// TIA Portal V20 export
TYPE "HMI_MotSpdL"
   STRUCT
      Spd1Man : Bool := FALSE;   // 1=Start: Speed1 Command in Manual Mode
      Spd2Man : Bool := FALSE;   // 1=Start: Speed2 Command in Manual Mode
      StopMan : Bool := FALSE;   // 1=Stop: Stop Command in Manual Mode
      AutModOp : Bool := FALSE;   // 1=Auto Mode: Auto Mode by Operator
      ManModOp : Bool := TRUE;   // 1=Manual Mode: Manual Mode by Operator
      LocalLi : Bool;   // 1=Local Mode: Local Operation by Field Signal
      LocalOp : Bool := FALSE;   // 1=Local Mode: Local Operation by Operator
      OosOp : Bool := FALSE;   // 1=Oos Mode: Oos Mode by Operator
      Spd1Local : Bool;   // 1=Start Local: Field Speed1 Start Signal
      Spd2Local : Bool;   // 1=Start Local: Field Speed2 Start Signal
      StopLocal : Bool;   // 1=Stop Local: Field Stop Signal
      Monitor : Bool := TRUE;   // 1=Monitor ON, 0=Monitor OFF: Feedback Monitor
      MonTiStatic : Real := 3.0;   // Monitoring Time of Feedback [s]
      MonTiDynamic : Real := 3.0;   // Monitoring Time of Feedback on starting or on change in control output [s]
      MonTiDyStop : Real := 3.0;   // Monitoring Time of Feedback on stopping in control output [s]
      RapidStp : Bool := FALSE;   // 1 = Motor Rapid Stop command
      RstOp : Bool := FALSE;   // Operator Reset Signal
      Permit_ST : Byte := BYTE#16#FF;   // Permit Signal Status
      PermSp2 : Bool := true;   // 1= Activation Speed2 is allowed, 0= Not allowed
      PermSp2_ST : Byte := BYTE#16#FF;   // PermSp2 Signal Status
      Intlock_ST : Byte := BYTE#16#FF;   // Interlock Signal Status
      IntlSp2 : Bool := true;   // 0= Intlock Speed2 is active, 1= Not active
      IntlSp2_ST : Byte := BYTE#16#FF;   // IntlSp2 Signal Status
      Protect_ST : Byte := BYTE#16#FF;   // Protect Signal Status
      ProtSp2 : Bool := true;   // 0= Protection Speed2 is active, 1= Not active
      ProtSp2_ST : Byte := BYTE#16#FF;   // ProtSp2 Signal Status
      UserAna1 : Real;   // User Analog Input 1
      UA1unit : Int := 0;   // Unit of UserAna1
      UserAna2 : Real;   // User Analog Input 2
      UA2unit : Int := 0;   // Unit of UserAna2
      BatchID : DWord := 16#0;   // Current Batch ID (number)
      BatchName : String[32] := '';   // Current Batch Name
      StepNo : DWord := 16#0;   // Batch Step Number
      CurrMon { ExternalWritable := 'False'} : DInt := 0;   // Remaining monitoring time [s]
      FbkSpd1Out { ExternalWritable := 'False'} : Bool;   // 1=Speed1, 0=Stop: Feedback of Control Speed1
      FbkSpd2Out { ExternalWritable := 'False'} : Bool;   // 1=Speed2, 0=Stop: Feedback of Control Speed2
      OS_PermOut { ExternalWritable := 'False'} : DWord := DWORD#16#FFFF_FFFF;   // Operator Permission: Output for OS
      OS_PermLog { ExternalWritable := 'False'} : DWord := DWORD#16#FFFF_FFFF;   // Operator Permission: Output for OS
      OpSt_Out { ExternalWritable := 'False'} : DWord := 16#0;   // Enabled operator stations
      ST_Worst { ExternalWritable := 'False'} : Byte := 16#80;   // Worst Signal Status
      AutoST { ExternalWritable := 'False'} : Byte := 16#80;   // Worst Signal Status of the automatic commands
      Status1 { ExternalWritable := 'False'} : DWord := 16#0;   // Status1 Word
      Status2 { ExternalWritable := 'False'} : DWord := 16#0;   // Status2 Word
      Status3 { ExternalWritable := 'False'} : DWord := 16#0;   // Status3 Word
      Status4 { ExternalWritable := 'False'} : DWord := 16#0;   // Status4 Word
      Status5 { ExternalWritable := 'False'} : DWord := 16#0;   // Status5 Word
      AlarmState { ExternalWritable := 'False'} : Word;   // Alarm State for group display / Alarm Status for group display
   END_STRUCT;
END_TYPE
